Omron CX-Programmer project Projeto3_Estampadora (CX-Programmer 9.75)

# PLC PLC1: CJ2M CPU11
I/O table (CPU CJ2M-CPU11): rack 0 slot 0 CJ1W-ID211; rack 0 slot 1 CJ1W-OD211; rack 0 slot 2 CJ1W-DA021; rack 0 slot 3 CJ1W-AD041-V1

## Global symbols (name address type ; comment)
0.00 BOOL  ; Selec Auto/Manual
0.01 BOOL  ; Botão Start
0.02 BOOL  ; Botão Stop
0.03 BOOL  ; Emergência
0.04 BOOL  ; Emergência Variador
0.05 BOOL  ; Sensor de Posição Inicial
0.06 BOOL  ; Sensor de Posição 1 (Prensa)
0.07 BOOL  ; Sensor de Posição 2 (Inspeção)
0.08 BOOL  ; Sensor de Posição 3 (Fim)
0.09 BOOL  ; Pneum_Ext
0.10 BOOL  ; Pneum_Retraido
0.11 BOOL  ; Sinal Inspeção OK
0.12 BOOL  ; Sinal Inspeção NOK
0.13 BOOL  ; Confirmação Remoção de Peça
0.14 BOOL  ; Sensor Servo +
0.15 BOOL  ; Sensor Servo-
1.00 BOOL  ; Luz de Aviso Vermelha
1.01 BOOL  ; Desligar Visão
1.02 BOOL  ; Luz de Aviso Amarela
1.03 BOOL  ; Luz de Funcionamento Verde
1.04 BOOL  ; Contactor Avanço do Motor
1.05 BOOL  ; Acionamento Visão
1.06 BOOL  ; Contactor Marcha-Atrás do Motor
1.07 BOOL  ; Válvula Pneumática - Estender
1.08 BOOL  ; Válvula Pneumática - Retrair
1.09 BOOL  ; Led Camara
1.10 BOOL  ; Sinal Robot 1
1.11 BOOL  ; Sinal Robot 2
1.12 BOOL  ; Servo Motor -
1.13 BOOL  ; Servo Motor +
1.14 BOOL  ; RESERVADO
1.15 BOOL  ; RESERVADO
30.00 BOOL  ; Relay_Aux
C0 CHANNEL  ; Contador peças OK
C0002 BOOL  ; Contador Alarme NOK
C1 CHANNEL  ; Contador peças NOK
D0 CHANNEL  ; Controlo Modo Automatico
D1 CHANNEL  ; Controlo Modo Manual
D10 CHANNEL  ; Etapa
D100 CHANNEL  ; Dados IHM Etapas Automáticas
D101 CHANNEL  ; Dados IHM Contador peças OK
D102 CHANNEL  ; Dados IHM Contador peças NOK
D103 CHANNEL  ; Dados IHM Modo Manual
D2 CHANNEL  ; Controlo Fim de Ciclo
T0000 BOOL  ; Temp_press
T0001 BOOL  ; Temp_NOK
T0002 BOOL  ; Temp_Visão
T0003 BOOL  ; Temp_Fim_Visão
T0004 BOOL  ; Timer Alarme 1
T0005 BOOL  ; Timer Alame 2
T0006 BOOL  ; Timer Alarme 3
T0007 BOOL  ; Timer Alarme 4
T0008 BOOL  ; Timer Alarme 5
T0009 BOOL  ; Timer Alarme 6
W0.00 BOOL  ; Flag de Reset do Sistema
W0.01 BOOL  ; IHM Comando Manual Motor Avanço
W0.02 BOOL  ; IHM Comando Manual Motor Marcha-Atrás
W0.03 BOOL  ; IHM Comando Manual Estender Pneumático
W0.04 BOOL  ; IHM Comando Manual Retrair Pneumático
W0.05 BOOL  ; IHM Comando Manual Reset Contador
W0.06 BOOL  ; IHM Comando Manual Led Camara
W0.07 BOOL  ; IHM Emergencia
W0.08 BOOL  ; Manual Motor Avançar
W0.09 BOOL  ; Manual Motor Retroceder
W0.10 BOOL  ; Manual Valvula Estender
W0.11 BOOL  ; Manual Valvula Retrair
W0.12 BOOL  ; Manual Led Camara
W0.13 BOOL  ; Stop Ciclo
W0.15 BOOL  ; Controlo Modo Manual
W10.00 BOOL  ; IHM Start
W10.01 BOOL  ; IHM Stop
W10.02 BOOL  ; IHM NOK
W10.03 BOOL  ; IHM OK
W10.04 BOOL  ; Robot 2 Fim
W10.05 BOOL  ; Robot 1 Inicio
W10.06 BOOL  ; Robot Estampagem
W1.00 BOOL  ; IHM Contador Ciclo
W1.01 BOOL  ; IHM Contador_OK
W1.02 BOOL  ; IHM Contador_NOK
W1.03 BOOL  ; IHM Contador_Total
W1.04 BOOL  ; IHM Reset Contador Nok Max
W1.05 BOOL  ; Manual Servomotor +
W1.06 BOOL  ; Manual Servomotor -
W1.07 BOOL  ; IHM Comando manual Servomotor +
W1.08 BOOL  ; IHM Comando manual Servomotor -
W22.01 BOOL  ; Alm Inicio
W22.02 BOOL  ; Alm Pneumatico +
W22.03 BOOL  ; Alm Pneumatico -
W22.04 BOOL  ; Alm Visao
W22.05 BOOL  ; Alm Final
W22.06 BOOL  ; Alm Outtime
W22.07 BOOL  ; Alm Geral
W22.08 BOOL  ; Alm Contador Nok Max

## Program Controlo_Processo (cyclic task 0)
Local symbols
DO CHANNEL

### Section Inicializacao

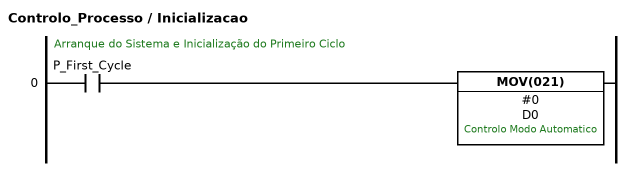
; rung 0: Arranque do Sistema e Inicialização do Primeiro Ciclo
LD P_First_Cycle
MOV(021) #0 D0  ; Controlo Modo Automatico

### Section Etapas
; Etapa 0: Inicialização e Verificação do Sistema

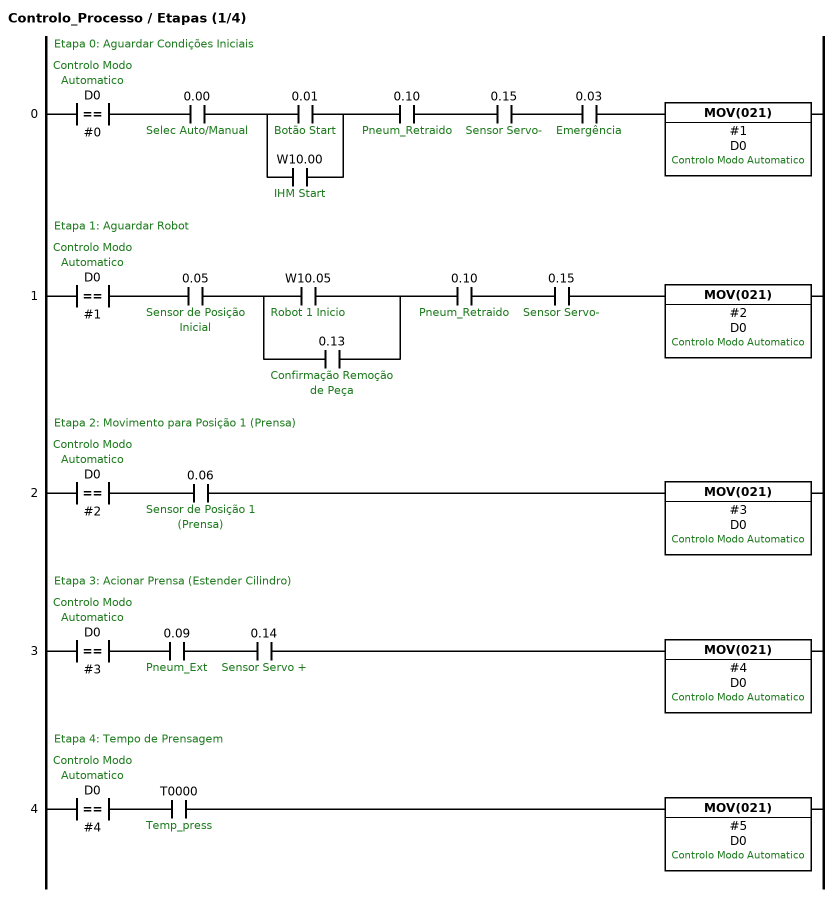
; rung 0: Etapa 0: Aguardar Condições Iniciais
LD=(300) D0 #0  ; Controlo Modo Automatico
AND 0.00  ; Selec Auto/Manual
LD 0.01  ; Botão Start
OR W10.00  ; IHM Start
ANDLD
AND 0.10  ; Pneum_Retraido
AND 0.15  ; Sensor Servo-
AND 0.03  ; Emergência
MOV(021) #1 D0  ; Controlo Modo Automatico
; rung 1: Etapa 1: Aguardar Robot
LD=(300) D0 #1  ; Controlo Modo Automatico
AND 0.05  ; Sensor de Posição Inicial
LD W10.05  ; Robot 1 Inicio
OR 0.13  ; Confirmação Remoção de Peça
ANDLD
AND 0.10  ; Pneum_Retraido
AND 0.15  ; Sensor Servo-
MOV(021) #2 D0  ; Controlo Modo Automatico
; rung 2: Etapa 2: Movimento para Posição 1 (Prensa)
LD=(300) D0 #2  ; Controlo Modo Automatico
AND 0.06  ; Sensor de Posição 1 (Prensa)
MOV(021) #3 D0  ; Controlo Modo Automatico
; rung 3: Etapa 3: Acionar Prensa (Estender Cilindro)
LD=(300) D0 #3  ; Controlo Modo Automatico
AND 0.09  ; Pneum_Ext
AND 0.14  ; Sensor Servo +
MOV(021) #4 D0  ; Controlo Modo Automatico
; rung 4: Etapa 4: Tempo de Prensagem
LD=(300) D0 #4  ; Controlo Modo Automatico
AND T0000  ; Temp_press
MOV(021) #5 D0  ; Controlo Modo Automatico

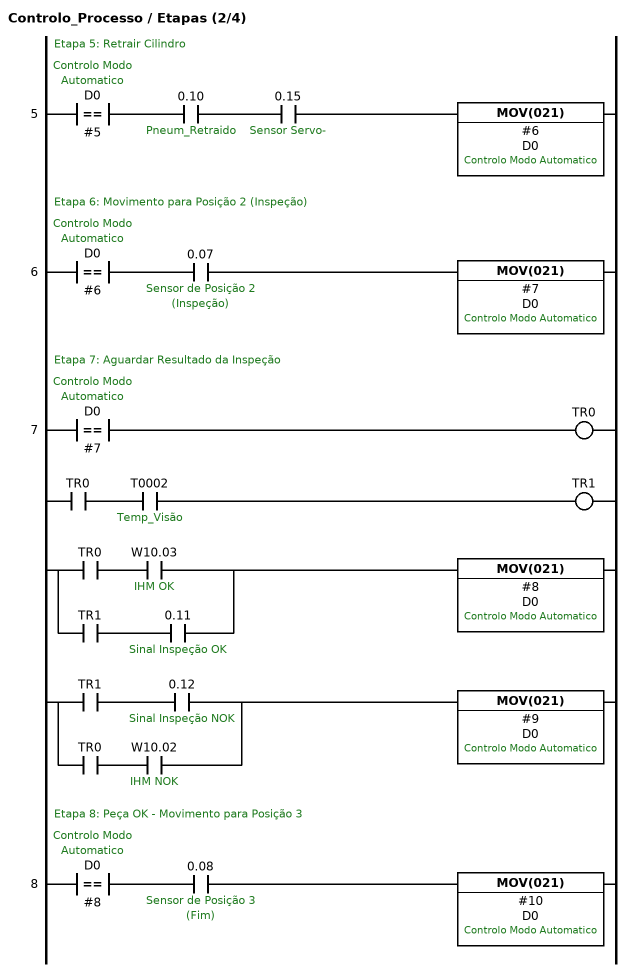
; rung 5: Etapa 5: Retrair Cilindro
LD=(300) D0 #5  ; Controlo Modo Automatico
AND 0.10  ; Pneum_Retraido
AND 0.15  ; Sensor Servo-
MOV(021) #6 D0  ; Controlo Modo Automatico
; rung 6: Etapa 6: Movimento para Posição 2 (Inspeção)
LD=(300) D0 #6  ; Controlo Modo Automatico
AND 0.07  ; Sensor de Posição 2 (Inspeção)
MOV(021) #7 D0  ; Controlo Modo Automatico
; rung 7: Etapa 7: Aguardar Resultado da Inspeção
LD=(300) D0 #7  ; Controlo Modo Automatico
OUT TR0
AND W10.03  ; IHM OK
LD TR0
AND T0002  ; Temp_Visão
OUT TR1
AND 0.11  ; Sinal Inspeção OK
ORLD
MOV(021) #8 D0  ; Controlo Modo Automatico
LD TR1
AND 0.12  ; Sinal Inspeção NOK
LD TR0
AND W10.02  ; IHM NOK
ORLD
MOV(021) #9 D0  ; Controlo Modo Automatico
; rung 8: Etapa 8: Peça OK - Movimento para Posição 3
LD=(300) D0 #8  ; Controlo Modo Automatico
AND 0.08  ; Sensor de Posição 3 (Fim)
MOV(021) #10 D0  ; Controlo Modo Automatico

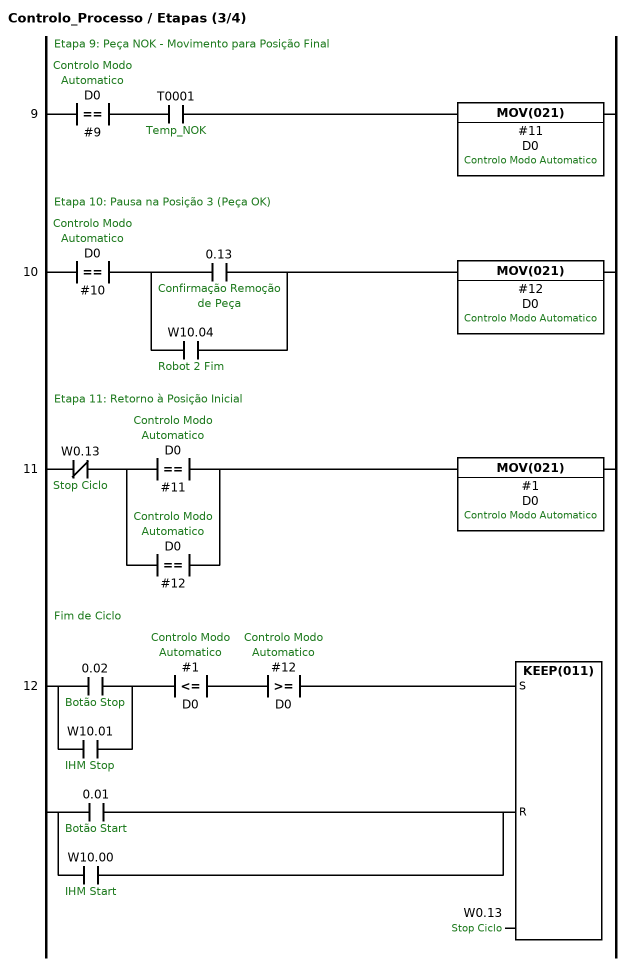
; rung 9: Etapa 9: Peça NOK - Movimento para Posição Final
LD=(300) D0 #9  ; Controlo Modo Automatico
AND T0001  ; Temp_NOK
MOV(021) #11 D0  ; Controlo Modo Automatico
; rung 10: Etapa 10: Pausa na Posição 3 (Peça OK)
LD=(300) D0 #10  ; Controlo Modo Automatico
LD 0.13  ; Confirmação Remoção de Peça
OR W10.04  ; Robot 2 Fim
ANDLD
MOV(021) #12 D0  ; Controlo Modo Automatico
; rung 11: Etapa 11: Retorno à Posição Inicial
LDNOT W0.13  ; Stop Ciclo
LD=(300) D0 #11  ; Controlo Modo Automatico
OR=(300) D0 #12  ; Controlo Modo Automatico
ANDLD
MOV(021) #1 D0  ; Controlo Modo Automatico
; rung 12: Fim de Ciclo
LD 0.02  ; Botão Stop
OR W10.01  ; IHM Stop
AND<=(315) #1 D0  ; Controlo Modo Automatico
AND>=(325) #12 D0  ; Controlo Modo Automatico
LD 0.01  ; Botão Start
OR W10.00  ; IHM Start
KEEP(011) W0.13  ; Stop Ciclo

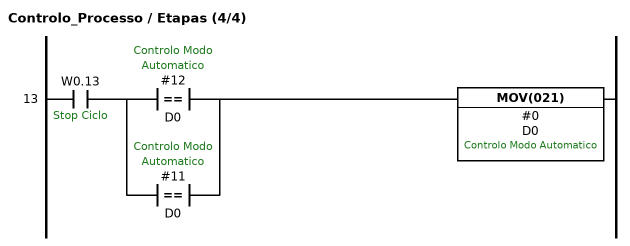
; rung 13
LD W0.13  ; Stop Ciclo
LD=(300) #12 D0  ; Controlo Modo Automatico
OR=(300) #11 D0  ; Controlo Modo Automatico
ANDLD
MOV(021) #0 D0  ; Controlo Modo Automatico

### Section Modo_Manual

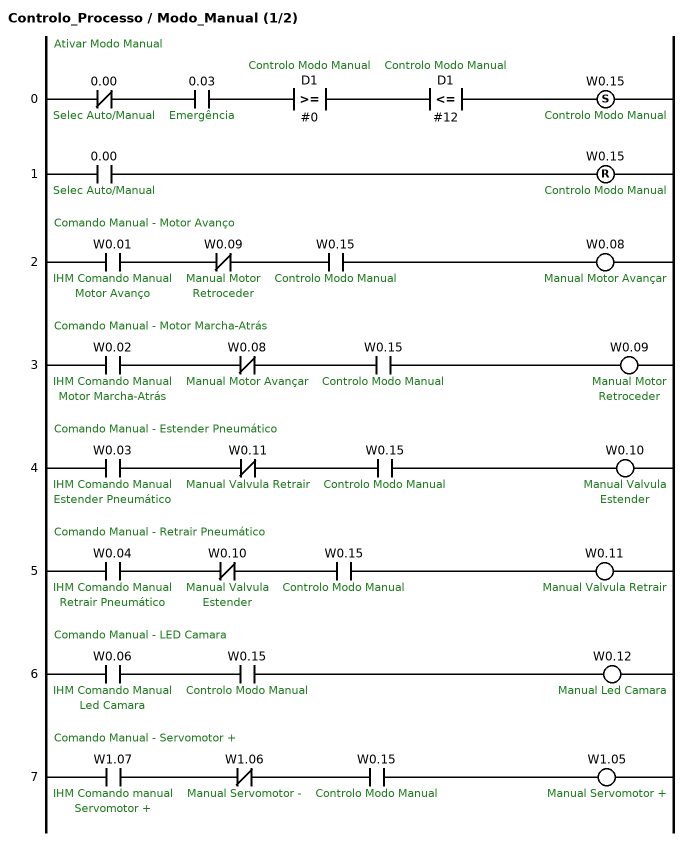
; rung 0: Ativar Modo Manual
LDNOT 0.00  ; Selec Auto/Manual
AND 0.03  ; Emergência
AND>=(325) D1 #0  ; Controlo Modo Manual
AND<=(315) D1 #12  ; Controlo Modo Manual
SET W0.15  ; Controlo Modo Manual
; rung 1
LD 0.00  ; Selec Auto/Manual
RSET W0.15  ; Controlo Modo Manual
; rung 2: Comando Manual - Motor Avanço
LD W0.01  ; IHM Comando Manual Motor Avanço
ANDNOT W0.09  ; Manual Motor Retroceder
AND W0.15  ; Controlo Modo Manual
OUT W0.08  ; Manual Motor Avançar
; rung 3: Comando Manual - Motor Marcha-Atrás
LD W0.02  ; IHM Comando Manual Motor Marcha-Atrás
ANDNOT W0.08  ; Manual Motor Avançar
AND W0.15  ; Controlo Modo Manual
OUT W0.09  ; Manual Motor Retroceder
; rung 4: Comando Manual - Estender Pneumático
LD W0.03  ; IHM Comando Manual Estender Pneumático
ANDNOT W0.11  ; Manual Valvula Retrair
AND W0.15  ; Controlo Modo Manual
OUT W0.10  ; Manual Valvula Estender
; rung 5: Comando Manual - Retrair Pneumático
LD W0.04  ; IHM Comando Manual Retrair Pneumático
ANDNOT W0.10  ; Manual Valvula Estender
AND W0.15  ; Controlo Modo Manual
OUT W0.11  ; Manual Valvula Retrair
; rung 6: Comando Manual - LED Camara
LD W0.06  ; IHM Comando Manual Led Camara
AND W0.15  ; Controlo Modo Manual
OUT W0.12  ; Manual Led Camara
; rung 7: Comando Manual - Servomotor +
LD W1.07  ; IHM Comando manual Servomotor +
ANDNOT W1.06  ; Manual Servomotor -
AND W0.15  ; Controlo Modo Manual
OUT W1.05  ; Manual Servomotor +

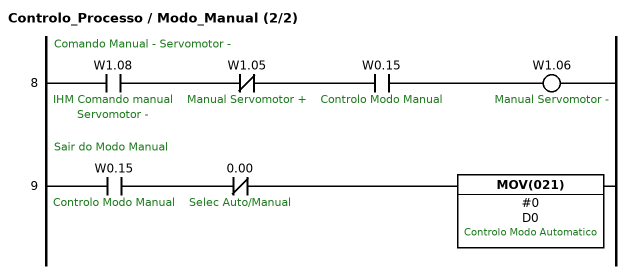
; rung 8: Comando Manual - Servomotor -
LD W1.08  ; IHM Comando manual Servomotor -
ANDNOT W1.05  ; Manual Servomotor +
AND W0.15  ; Controlo Modo Manual
OUT W1.06  ; Manual Servomotor -
; rung 9: Sair do Modo Manual
LD W0.15  ; Controlo Modo Manual
ANDNOT 0.00  ; Selec Auto/Manual
MOV(021) #0 D0  ; Controlo Modo Automatico

### Section Emergencia

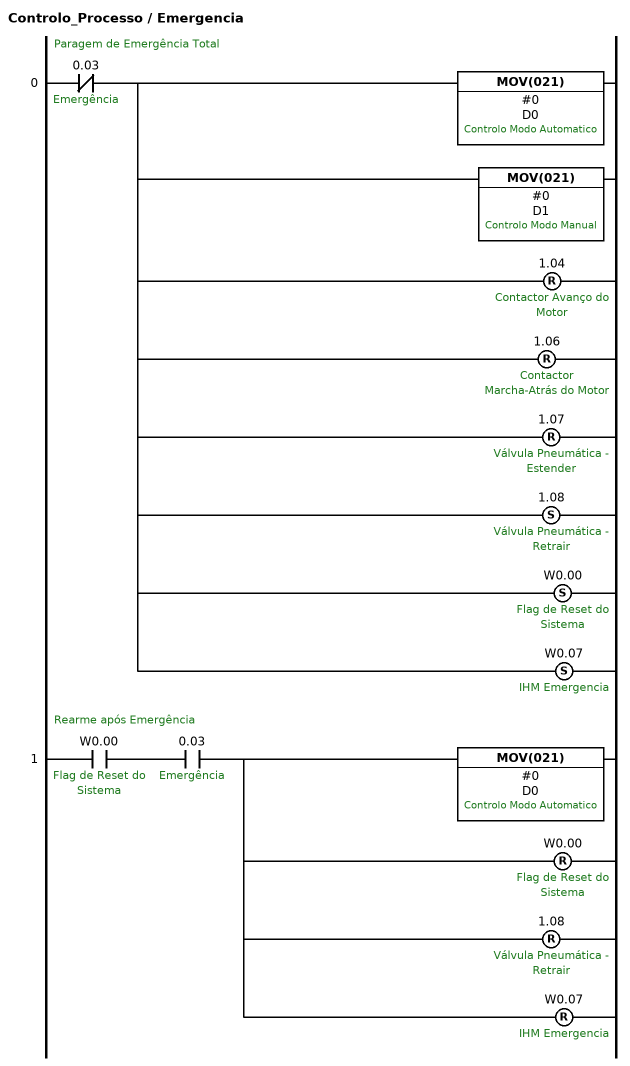
; rung 0: Paragem de Emergência Total
LDNOT 0.03  ; Emergência
MOV(021) #0 D0  ; Controlo Modo Automatico
MOV(021) #0 D1  ; Controlo Modo Manual
RSET 1.04  ; Contactor Avanço do Motor
RSET 1.06  ; Contactor Marcha-Atrás do Motor
RSET 1.07  ; Válvula Pneumática - Estender
SET 1.08  ; Válvula Pneumática - Retrair
SET W0.00  ; Flag de Reset do Sistema
SET W0.07  ; IHM Emergencia
; rung 1: Rearme após Emergência
LD W0.00  ; Flag de Reset do Sistema
AND 0.03  ; Emergência
MOV(021) #0 D0  ; Controlo Modo Automatico
RSET W0.00  ; Flag de Reset do Sistema
RSET 1.08  ; Válvula Pneumática - Retrair
RSET W0.07  ; IHM Emergencia

### Section Saidas_Motor

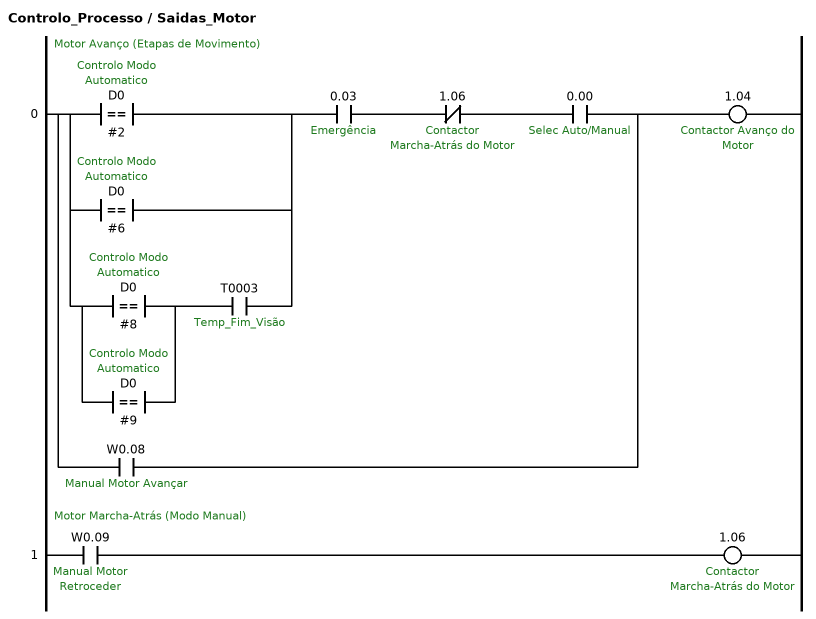
; rung 0: Motor Avanço (Etapas de Movimento)
LD=(300) D0 #2  ; Controlo Modo Automatico
OR=(300) D0 #6  ; Controlo Modo Automatico
LD=(300) D0 #8  ; Controlo Modo Automatico
OR=(300) D0 #9  ; Controlo Modo Automatico
AND T0003  ; Temp_Fim_Visão
ORLD
AND 0.03  ; Emergência
ANDNOT 1.06  ; Contactor Marcha-Atrás do Motor
AND 0.00  ; Selec Auto/Manual
OR W0.08  ; Manual Motor Avançar
OUT 1.04  ; Contactor Avanço do Motor
; rung 1: Motor Marcha-Atrás (Modo Manual)
LD W0.09  ; Manual Motor Retroceder
OUT 1.06  ; Contactor Marcha-Atrás do Motor

### Section Saidas_Pneumatico

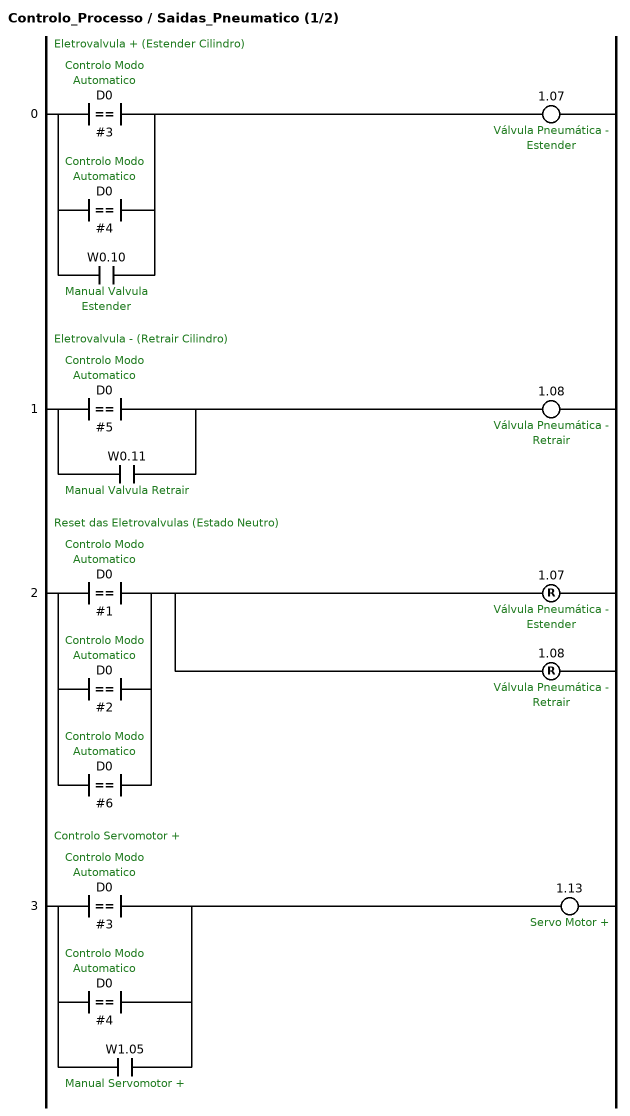
; rung 0: Eletrovalvula + (Estender Cilindro)
LD=(300) D0 #3  ; Controlo Modo Automatico
OR=(300) D0 #4  ; Controlo Modo Automatico
OR W0.10  ; Manual Valvula Estender
OUT 1.07  ; Válvula Pneumática - Estender
; rung 1: Eletrovalvula - (Retrair Cilindro)
LD=(300) D0 #5  ; Controlo Modo Automatico
OR W0.11  ; Manual Valvula Retrair
OUT 1.08  ; Válvula Pneumática - Retrair
; rung 2: Reset das Eletrovalvulas (Estado Neutro)
LD=(300) D0 #1  ; Controlo Modo Automatico
OR=(300) D0 #2  ; Controlo Modo Automatico
OR=(300) D0 #6  ; Controlo Modo Automatico
RSET 1.07  ; Válvula Pneumática - Estender
RSET 1.08  ; Válvula Pneumática - Retrair
; rung 3: Controlo Servomotor +
LD=(300) D0 #3  ; Controlo Modo Automatico
OR=(300) D0 #4  ; Controlo Modo Automatico
OR W1.05  ; Manual Servomotor +
OUT 1.13  ; Servo Motor +

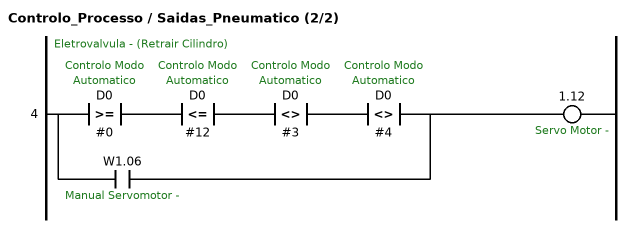
; rung 4: Eletrovalvula - (Retrair Cilindro)
LD>=(325) D0 #0  ; Controlo Modo Automatico
AND<=(315) D0 #12  ; Controlo Modo Automatico
AND<>(305) D0 #3  ; Controlo Modo Automatico
AND<>(305) D0 #4  ; Controlo Modo Automatico
OR W1.06  ; Manual Servomotor -
OUT 1.12  ; Servo Motor -

### Section Saidas_Sinalizacao

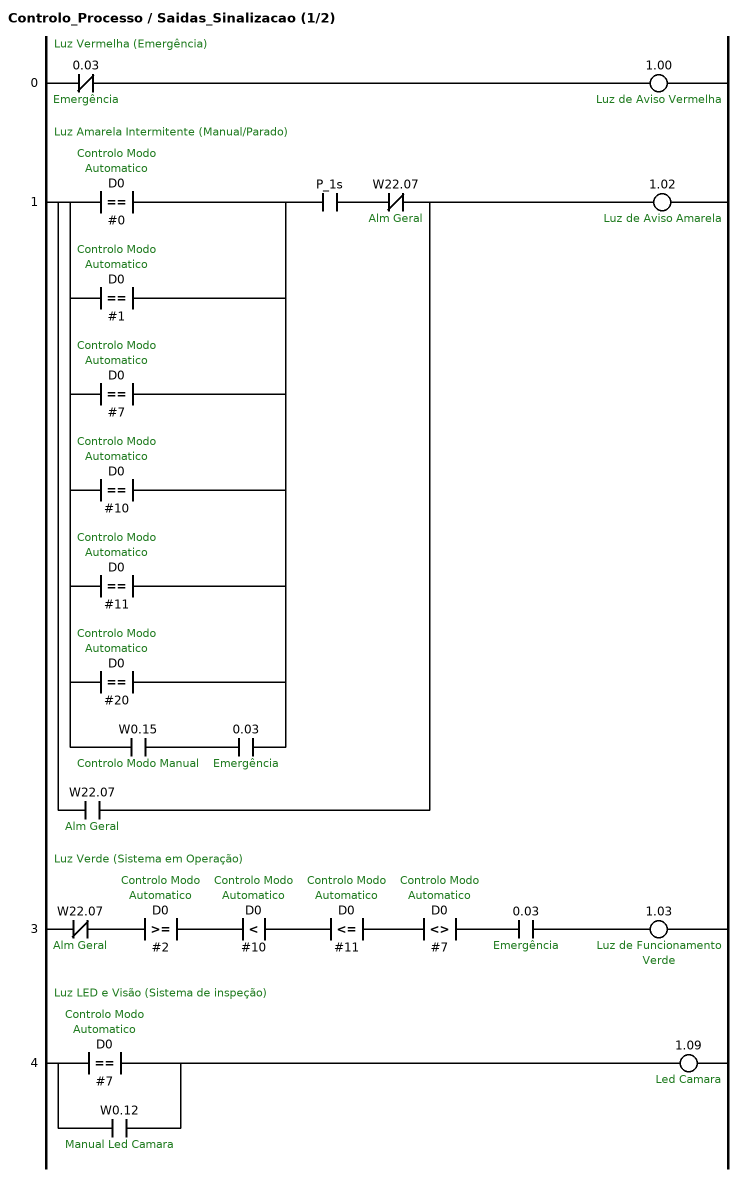
; rung 0: Luz Vermelha (Emergência)
LDNOT 0.03  ; Emergência
OUT 1.00  ; Luz de Aviso Vermelha
; rung 1: Luz Amarela Intermitente (Manual/Parado)
LD=(300) D0 #0  ; Controlo Modo Automatico
OR=(300) D0 #1  ; Controlo Modo Automatico
OR=(300) D0 #7  ; Controlo Modo Automatico
OR=(300) D0 #10  ; Controlo Modo Automatico
OR=(300) D0 #11  ; Controlo Modo Automatico
OR=(300) D0 #20  ; Controlo Modo Automatico
LD W0.15  ; Controlo Modo Manual
AND 0.03  ; Emergência
ORLD
AND P_1s
ANDNOT W22.07  ; Alm Geral
OR W22.07  ; Alm Geral
OUT 1.02  ; Luz de Aviso Amarela
; rung 3: Luz Verde (Sistema em Operação)
LDNOT W22.07  ; Alm Geral
AND>=(325) D0 #2  ; Controlo Modo Automatico
AND<(310) D0 #10  ; Controlo Modo Automatico
AND<=(315) D0 #11  ; Controlo Modo Automatico
AND<>(305) D0 #7  ; Controlo Modo Automatico
AND 0.03  ; Emergência
OUT 1.03  ; Luz de Funcionamento Verde
; rung 4: Luz LED e Visão (Sistema de inspeção)
LD=(300) D0 #7  ; Controlo Modo Automatico
OR W0.12  ; Manual Led Camara
OUT 1.09  ; Led Camara

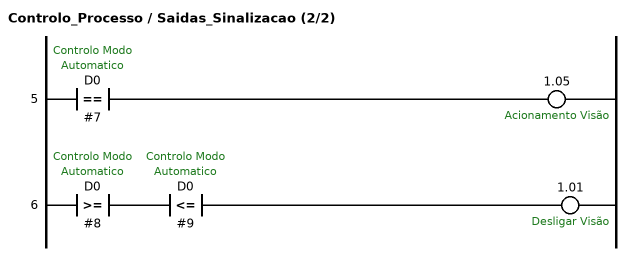
; rung 5
LD=(300) D0 #7  ; Controlo Modo Automatico
OUT 1.05  ; Acionamento Visão
; rung 6
LD>=(325) D0 #8  ; Controlo Modo Automatico
AND<=(315) D0 #9  ; Controlo Modo Automatico
OUT 1.01  ; Desligar Visão

### Section Saida_Robot

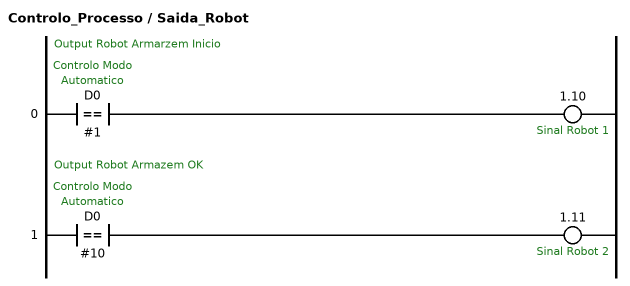
; rung 0: Output Robot Armarzem Inicio
LD=(300) D0 #1  ; Controlo Modo Automatico
OUT 1.10  ; Sinal Robot 1
; rung 1: Output Robot Armazem OK
LD=(300) D0 #10  ; Controlo Modo Automatico
OUT 1.11  ; Sinal Robot 2

### Section Temporizadores

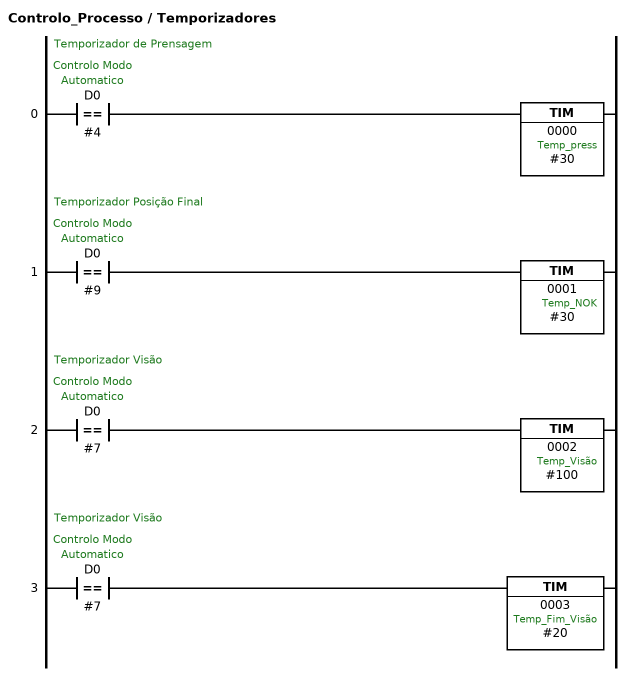
; rung 0: Temporizador de Prensagem
LD=(300) D0 #4  ; Controlo Modo Automatico
TIM 0000 #30  ; Temp_press
; rung 1: Temporizador Posição Final
LD=(300) D0 #9  ; Controlo Modo Automatico
TIM 0001 #30  ; Temp_NOK
; rung 2: Temporizador Visão
LD=(300) D0 #7  ; Controlo Modo Automatico
TIM 0002 #100  ; Temp_Visão
; rung 3: Temporizador Visão
LD=(300) D0 #7  ; Controlo Modo Automatico
TIM 0003 #20  ; Temp_Fim_Visão

### Section Contadores

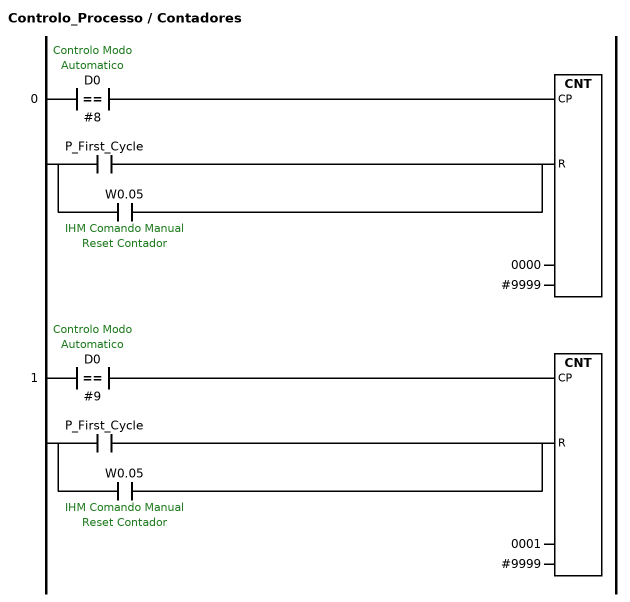
; rung 0
LD=(300) D0 #8  ; Controlo Modo Automatico
LD P_First_Cycle
OR W0.05  ; IHM Comando Manual Reset Contador
CNT 0000 #9999
; rung 1
LD=(300) D0 #9  ; Controlo Modo Automatico
LD P_First_Cycle
OR W0.05  ; IHM Comando Manual Reset Contador
CNT 0001 #9999

### Section IHM_Alarmes

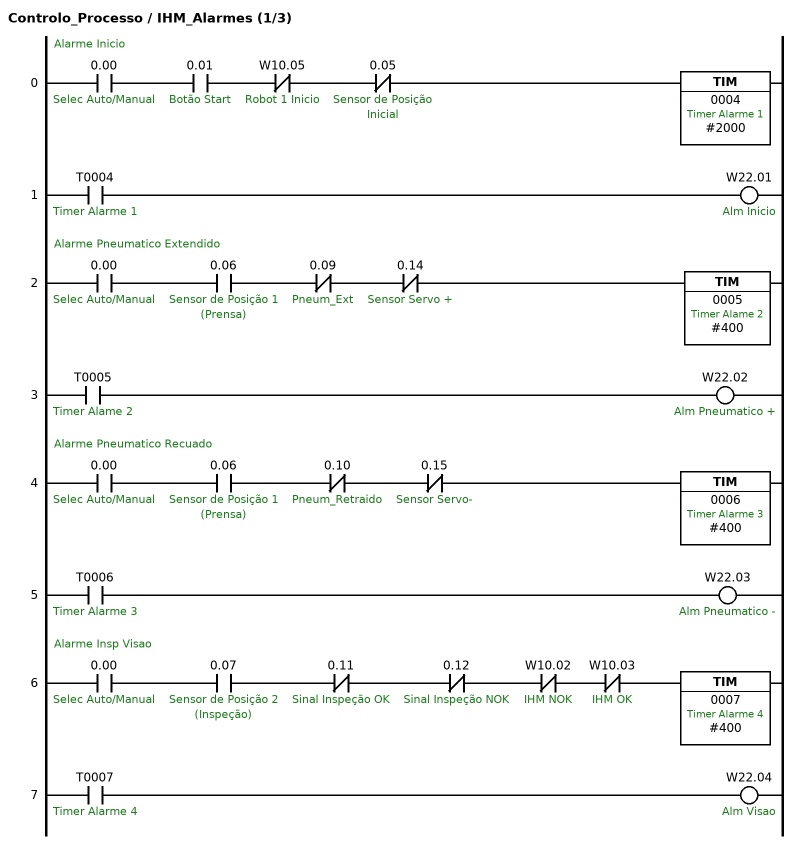
; rung 0: Alarme Inicio
LD 0.00  ; Selec Auto/Manual
AND 0.01  ; Botão Start
ANDNOT W10.05  ; Robot 1 Inicio
ANDNOT 0.05  ; Sensor de Posição Inicial
TIM 0004 #2000  ; Timer Alarme 1
; rung 1
LD T0004  ; Timer Alarme 1
OUT W22.01  ; Alm Inicio
; rung 2: Alarme Pneumatico Extendido
LD 0.00  ; Selec Auto/Manual
AND 0.06  ; Sensor de Posição 1 (Prensa)
ANDNOT 0.09  ; Pneum_Ext
ANDNOT 0.14  ; Sensor Servo +
TIM 0005 #400  ; Timer Alame 2
; rung 3
LD T0005  ; Timer Alame 2
OUT W22.02  ; Alm Pneumatico +
; rung 4: Alarme Pneumatico Recuado
LD 0.00  ; Selec Auto/Manual
AND 0.06  ; Sensor de Posição 1 (Prensa)
ANDNOT 0.10  ; Pneum_Retraido
ANDNOT 0.15  ; Sensor Servo-
TIM 0006 #400  ; Timer Alarme 3
; rung 5
LD T0006  ; Timer Alarme 3
OUT W22.03  ; Alm Pneumatico -
; rung 6: Alarme Insp Visao
LD 0.00  ; Selec Auto/Manual
AND 0.07  ; Sensor de Posição 2 (Inspeção)
ANDNOT 0.11  ; Sinal Inspeção OK
ANDNOT 0.12  ; Sinal Inspeção NOK
ANDNOT W10.02  ; IHM NOK
ANDNOT W10.03  ; IHM OK
TIM 0007 #400  ; Timer Alarme 4
; rung 7
LD T0007  ; Timer Alarme 4
OUT W22.04  ; Alm Visao

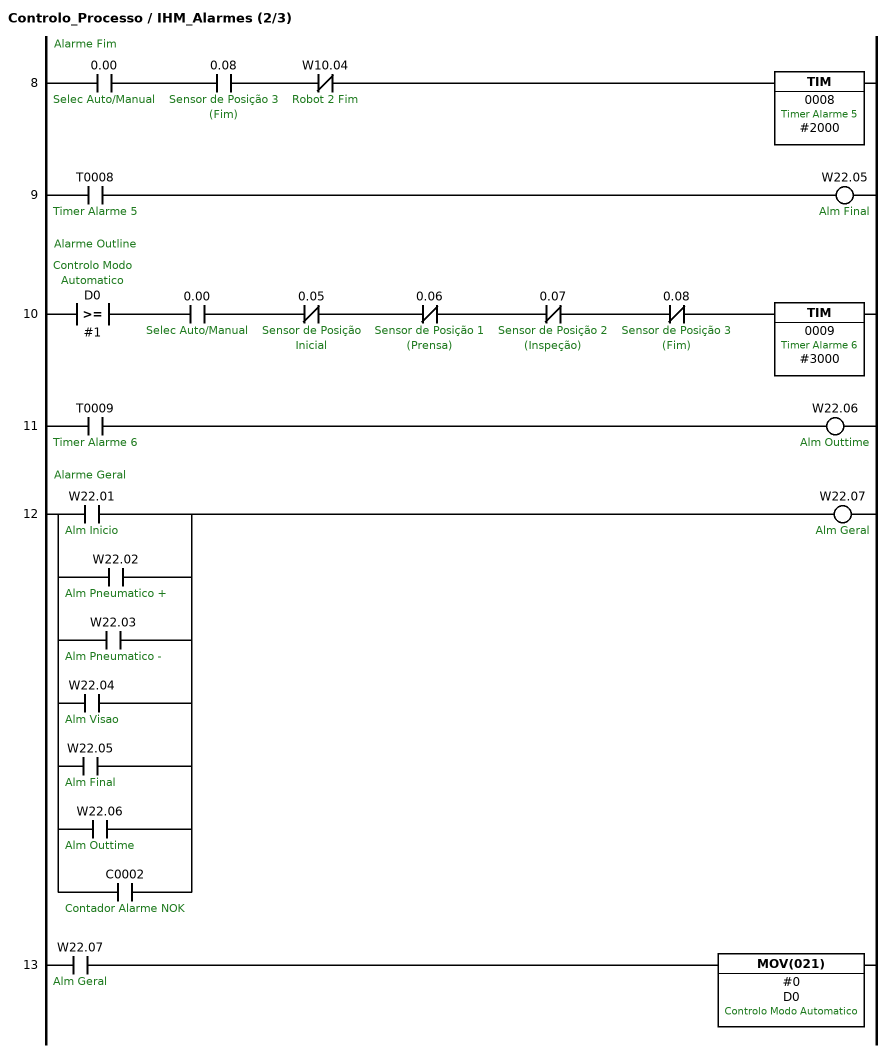
; rung 8: Alarme Fim
LD 0.00  ; Selec Auto/Manual
AND 0.08  ; Sensor de Posição 3 (Fim)
ANDNOT W10.04  ; Robot 2 Fim
TIM 0008 #2000  ; Timer Alarme 5
; rung 9
LD T0008  ; Timer Alarme 5
OUT W22.05  ; Alm Final
; rung 10: Alarme Outline
LD>=(325) D0 #1  ; Controlo Modo Automatico
AND 0.00  ; Selec Auto/Manual
ANDNOT 0.05  ; Sensor de Posição Inicial
ANDNOT 0.06  ; Sensor de Posição 1 (Prensa)
ANDNOT 0.07  ; Sensor de Posição 2 (Inspeção)
ANDNOT 0.08  ; Sensor de Posição 3 (Fim)
TIM 0009 #3000  ; Timer Alarme 6
; rung 11
LD T0009  ; Timer Alarme 6
OUT W22.06  ; Alm Outtime
; rung 12: Alarme Geral
LD W22.01  ; Alm Inicio
OR W22.02  ; Alm Pneumatico +
OR W22.03  ; Alm Pneumatico -
OR W22.04  ; Alm Visao
OR W22.05  ; Alm Final
OR W22.06  ; Alm Outtime
OR C0002  ; Contador Alarme NOK
OUT W22.07  ; Alm Geral
; rung 13
LD W22.07  ; Alm Geral
MOV(021) #0 D0  ; Controlo Modo Automatico

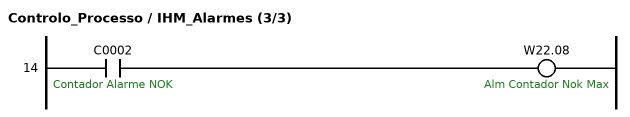
; rung 14
LD C0002  ; Contador Alarme NOK
OUT W22.08  ; Alm Contador Nok Max

### Section IHM_Interface

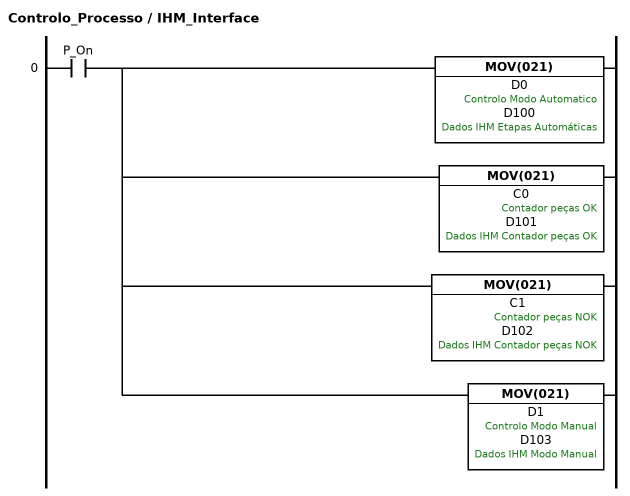
; rung 0
LD P_On
MOV(021) D0 D100  ; Controlo Modo Automatico, Dados IHM Etapas Automáticas
MOV(021) C0 D101  ; Contador peças OK, Dados IHM Contador peças OK
MOV(021) C1 D102  ; Contador peças NOK, Dados IHM Contador peças NOK
MOV(021) D1 D103  ; Controlo Modo Manual, Dados IHM Modo Manual

### Section IHM_Contadores_Temporizadores

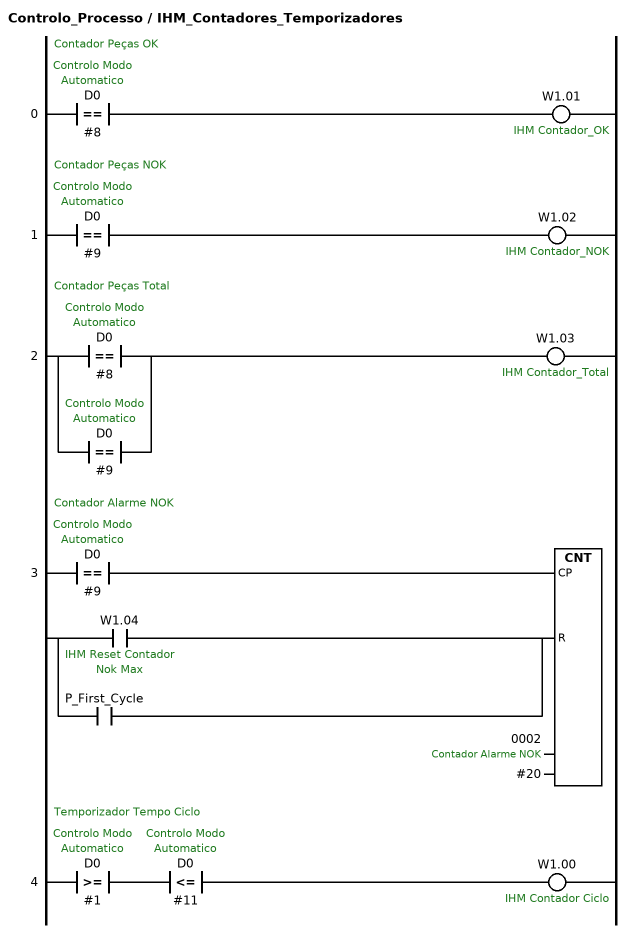
; rung 0: Contador Peças OK
LD=(300) D0 #8  ; Controlo Modo Automatico
OUT W1.01  ; IHM Contador_OK
; rung 1: Contador Peças NOK
LD=(300) D0 #9  ; Controlo Modo Automatico
OUT W1.02  ; IHM Contador_NOK
; rung 2: Contador Peças Total
LD=(300) D0 #8  ; Controlo Modo Automatico
OR=(300) D0 #9  ; Controlo Modo Automatico
OUT W1.03  ; IHM Contador_Total
; rung 3: Contador Alarme NOK
LD=(300) D0 #9  ; Controlo Modo Automatico
LD W1.04  ; IHM Reset Contador Nok Max
OR P_First_Cycle
CNT 0002 #20  ; Contador Alarme NOK
; rung 4: Temporizador Tempo Ciclo
LD>=(325) D0 #1  ; Controlo Modo Automatico
AND<=(315) D0 #11  ; Controlo Modo Automatico
OUT W1.00  ; IHM Contador Ciclo

### Section END
; rung 0
END(001)